// TIA Portal V21 export
FUNCTION "PassiProduzione_010102" : Void   // FC145, LAD
{ S7_Optimized_Access := 'TRUE' }
// stored: SetENOAutomatically false
   VAR_TEMP
      CondizioniPassoEsterne : Bool;
      AbilitazionePasso : Bool;
      AppoggioComando : Int;
      ComandoValvolaB : Int;
      PompaPistoniAbilitata : Bool;
   END_VAR
   VAR CONSTANT
      Positivo : Int := 2;
      Negativo : Int := 3;
      FolleScarico : Int := 4;
      FlipFlop : Int := 5;
      SmettiDiContare : Int := 0;
      ResettaIlConteggio : Int := 1;
      Stop : Int := 6;
   END_VAR
BEGIN

REGION Network 1: Sequenza: Produzione - Passo: Sterilizzazione. Condizioni passo esterne.
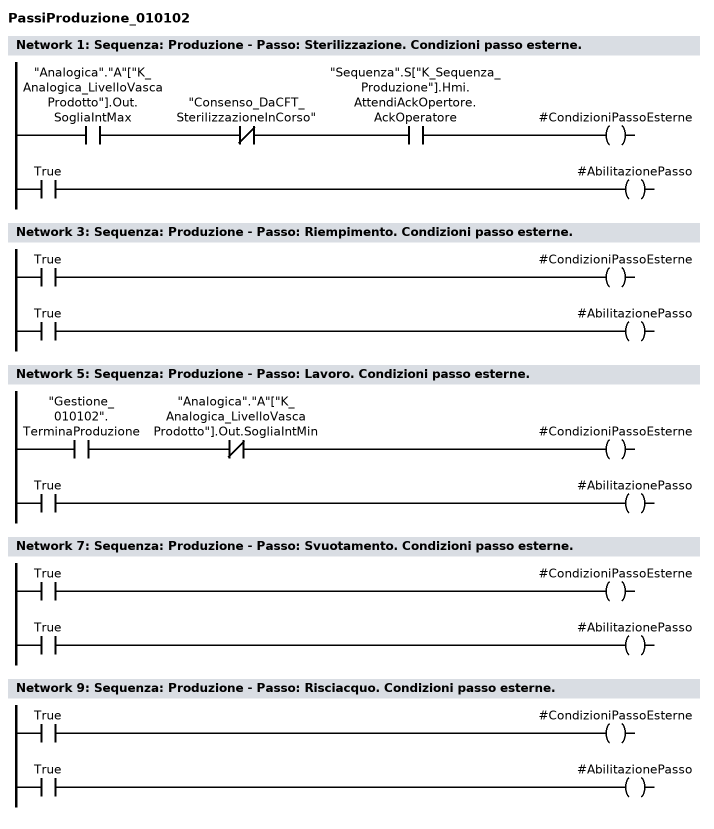
   RUNG wire#powerrail
      Contact( "Analogica"."A"["K_Analogica_LivelloVascaProdotto"].Out.SogliaIntMax )
      I_Contact( "Consenso_DaCFT_SterilizzazioneInCorso" )
      Contact( "Sequenza".S["K_Sequenza_Produzione"].Hmi.AttendiAckOpertore.AckOperatore )
      Coil( #CondizioniPassoEsterne )
   END_RUNG
   RUNG wire#powerrail
      Contact( True )
      Coil( #AbilitazionePasso )
   END_RUNG
   // the same network as SCL:
   #CondizioniPassoEsterne := "Analogica"."A"["K_Analogica_LivelloVascaProdotto"].Out.SogliaIntMax AND NOT "Consenso_DaCFT_SterilizzazioneInCorso" AND "Sequenza".S["K_Sequenza_Produzione"].Hmi.AttendiAckOpertore.AckOperatore;
   #AbilitazionePasso := True;
END_REGION

REGION Network 2 (SCL): Sequenza: Produzione - Passo: Sterilizzazione. Gestione del passo.
   REGION Parametri del passo
       "GestPasso"(K_PassoAttuale := "K_Passo_Sterilizzazione",
                   K_PassoSuccessivo := "K_Passo_Riempimento",
                   AbilitaSaltapasso := True,
                   AbilitaPasso:= #AbilitazionePasso,
                   CondizioniPassoEsterne := #CondizioniPassoEsterne,
                   K_Sequenza := "K_Sequenza_Produzione");
   END_REGION ;
   REGION Comando delle utenze nel passo 
       "GestPasso_CmdValvola"(K_Valvola := "K_Valvola_I",
                              Comando := #Positivo,
                              K_Sequenza := "K_Sequenza_Produzione",
                              K_Passo := "K_Passo_Sterilizzazione",
                              NonAttenderePosizione := False);

       "GestPasso_CmdValvola"(K_Valvola := "K_Valvola_D",
                              Comando := #Positivo,
                              K_Sequenza := "K_Sequenza_Produzione",
                              K_Passo := "K_Passo_Sterilizzazione",
                              NonAttenderePosizione := False);

       "GestPasso_CmdValvola"(K_Valvola := "K_Valvola_D2",
                              Comando := #Positivo,
                              K_Sequenza := "K_Sequenza_Produzione",
                              K_Passo := "K_Passo_Sterilizzazione",
                              NonAttenderePosizione := True);

       "GestPasso_CmdValvola"(K_Valvola := "K_Valvola_B",
                              Comando := #Positivo,
                              K_Sequenza := "K_Sequenza_Produzione",
                              K_Passo := "K_Passo_Sterilizzazione",
                              NonAttenderePosizione := False);

       "GestPasso_CmdValvola"(K_Valvola := "K_Valvola_B1",
                              Comando := "GestPasso_ReplicaComandoValvola"("K_Valvola_B"),
                              K_Sequenza := "K_Sequenza_Produzione",
                              K_Passo := "K_Passo_Sterilizzazione",
                              NonAttenderePosizione := False);

       "GestPasso_CmdValvolaFlipFlop"(K_Valvola := "K_Valvola_L",
                                      NumeroCicli := 1,
                                      TempoPositivo := 1500,
                                      TempoNegativo := 5,
                                      ComandoARiposo := #Negativo,
                                      K_Passo := "K_Passo_Sterilizzazione",
                                      K_Sequenza := "K_Sequenza_Produzione");

       "GestPasso_CmdValvola"(K_Valvola := "K_Valvola_F",
                              Comando := #Positivo,
                              K_Sequenza := "K_Sequenza_Produzione",
                              K_Passo := "K_Passo_Sterilizzazione",
                              NonAttenderePosizione := False);

       "GestPasso_CmdValvola"(K_Valvola := "K_Valvola_CP1",
                              Comando := #Positivo,
                              K_Sequenza := "K_Sequenza_Produzione",
                              K_Passo := "K_Passo_Sterilizzazione",
                              NonAttenderePosizione := False);

       "GestPasso_CmdValvola"(K_Valvola := "K_Valvola_CP2",
                              Comando := #Positivo,
                              K_Sequenza := "K_Sequenza_Produzione",
                              K_Passo := "K_Passo_Sterilizzazione",
                              NonAttenderePosizione := False);

       "GestPasso_AttendiAnalogica"(K_Analogica := "K_Analogica_TemperaturaFineLinea",
                                    KAllAnalog := "KAllAnalog_IntMax",
                                    Comportamento := #ResettaIlConteggio,
                                    K_Sequenza := "K_Sequenza_Produzione",
                                    K_Passo := "K_Passo_Sterilizzazione",
                                    NonAttenderePosizione := False);
       //Motori
       "GestPasso_CmdMotore"(K_Motore := "K_Motore_PompaRicircoloAcquaCalda",
                             Comando := #Positivo,
                             K_Sequenza := "K_Sequenza_Produzione",
                             K_Passo := "K_Passo_Sterilizzazione",
                             NonAttenderePosizione := False);
   END_REGION ;
END_REGION

REGION Network 3: Sequenza: Produzione - Passo: Riempimento. Condizioni passo esterne.
   RUNG wire#powerrail
      Contact( True )
      Coil( #CondizioniPassoEsterne )
   END_RUNG
   RUNG wire#powerrail
      Contact( True )
      Coil( #AbilitazionePasso )
   END_RUNG
   // the same network as SCL:
   #CondizioniPassoEsterne := True;
   #AbilitazionePasso := True;
END_REGION

REGION Network 4 (SCL): Sequenza: Produzione - Passo: Riempimento. Gestione del passo.
   REGION Parametri del passo
       "GestPasso"(K_PassoAttuale := "K_Passo_Riempimento",
                   K_PassoSuccessivo := "K_Passo_Lavoro",
                   AbilitaSaltapasso := True,
                   AbilitaPasso:= #AbilitazionePasso,
                   CondizioniPassoEsterne := #CondizioniPassoEsterne,
                   K_Sequenza := "K_Sequenza_Produzione");
   END_REGION ;
   REGION Comando delle utenze nel passo 

       "GestPasso_CmdValvola"(K_Valvola := "K_Valvola_D",
                              Comando := #Positivo,
                              K_Sequenza := "K_Sequenza_Produzione",
                              K_Passo := "K_Passo_Riempimento",
                              NonAttenderePosizione := False);

       "GestPasso_CmdValvola"(K_Valvola := "K_Valvola_D2",
                              Comando := #Positivo,
                              K_Sequenza := "K_Sequenza_Produzione",
                              K_Passo := "K_Passo_Riempimento",
                              NonAttenderePosizione := False);

       IF "Analogica".A[K_Analogica_TemperaturaUscitaSterilizzatoreProcesso].Out.SogliaIntMin THEN
           #ComandoValvolaB := #Positivo;
       ELSE
           #ComandoValvolaB := #Negativo;
       END_IF;

       "GestPasso_CmdValvola"(K_Valvola := "K_Valvola_R",
                              Comando := #Positivo,
                              K_Sequenza := "K_Sequenza_Produzione",
                              K_Passo := "K_Passo_Riempimento",
                              NonAttenderePosizione := False);

       "GestPasso_CmdValvola"(K_Valvola := "K_Valvola_B",
                              Comando := #ComandoValvolaB,
                              K_Sequenza := "K_Sequenza_Produzione",
                              K_Passo := "K_Passo_Riempimento",
                              NonAttenderePosizione := False);

       "GestPasso_CmdValvola"(K_Valvola := "K_Valvola_B1",
                              Comando := "GestPasso_ReplicaComandoValvola"("K_Valvola_B"),
                              K_Sequenza := "K_Sequenza_Produzione",
                              K_Passo := "K_Passo_Riempimento",
                              NonAttenderePosizione := False);

       "GestPasso_CmdValvola"(K_Valvola := "K_Valvola_CP1",
                              Comando := #Positivo,
                              K_Sequenza := "K_Sequenza_Produzione",
                              K_Passo := "K_Passo_Riempimento",
                              NonAttenderePosizione := False);

       "GestPasso_CmdValvola"(K_Valvola := "K_Valvola_CP2",
                              Comando := #Positivo,
                              K_Sequenza := "K_Sequenza_Produzione",
                              K_Passo := "K_Passo_Riempimento",
                              NonAttenderePosizione := False);

       "GestPasso_AttendiTotalizzatore"(K_Portata := "K_Portata_PortataIngresso",
                                        K_Sequenza := "K_Sequenza_Produzione",
                                        K_Passo := "K_Passo_Riempimento",
                                        NonAttenderePosizione := False,
                                        Preset_Metricubi := "Gestione_010102".MetricubiTubazioneRiempimento);


       //Motori
       "GestPasso_CmdMotore"(K_Motore := "K_Motore_PompaRicircoloAcquaCalda",
                             Comando := #Positivo,
                             K_Sequenza := "K_Sequenza_Produzione",
                             K_Passo := "K_Passo_Riempimento",
                             NonAttenderePosizione := False);

       #PompaPistoniAbilitata := "MacchinaARicetta".M[K_MacchinaARicetta_SterilizzatoreTubo].Lavoro.DatoBool[K_DatoRicettaBool_SterilizzatoreTubo_AbilitazionePompaPistoni];

       IF #PompaPistoniAbilitata THEN
           "GestPasso_CmdMotore"(K_Motore := "K_Motore_PompaPistoni",
                                 Comando := #Positivo,
                                 K_Sequenza := "K_Sequenza_Produzione",
                                 K_Passo := "K_Passo_Riempimento",
                                 NonAttenderePosizione := False);
       END_IF;
       "GestPasso_CmdMotore"(K_Motore := "K_Motore_PompaMono",
                             Comando := #Positivo,
                             K_Sequenza := "K_Sequenza_Produzione",
                             K_Passo := "K_Passo_Riempimento",
                             NonAttenderePosizione := False);
   END_REGION ;
END_REGION

REGION Network 5: Sequenza: Produzione - Passo: Lavoro. Condizioni passo esterne.
   RUNG wire#powerrail
      Contact( "Gestione_010102".TerminaProduzione )
      I_Contact( "Analogica"."A"["K_Analogica_LivelloVascaProdotto"].Out.SogliaIntMin )
      Coil( #CondizioniPassoEsterne )
   END_RUNG
   RUNG wire#powerrail
      Contact( True )
      Coil( #AbilitazionePasso )
   END_RUNG
   // the same network as SCL:
   #CondizioniPassoEsterne := "Gestione_010102".TerminaProduzione AND NOT "Analogica"."A"["K_Analogica_LivelloVascaProdotto"].Out.SogliaIntMin;
   #AbilitazionePasso := True;
END_REGION

REGION Network 6 (SCL): Sequenza: Produzione - Passo: Lavoro. Gestione del passo.
   REGION Parametri del passo
       "GestPasso"(K_PassoAttuale := "K_Passo_Lavoro",
                   K_PassoSuccessivo := "K_Passo_Svuotamento",
                   AbilitaSaltapasso := True,
                   AbilitaPasso:= #AbilitazionePasso,
                   CondizioniPassoEsterne := #CondizioniPassoEsterne,
                   K_Sequenza := "K_Sequenza_Produzione");
   END_REGION ;
   REGION Comando delle utenze nel passo 


       "GestPasso_CmdValvola"(K_Valvola := "K_Valvola_D",
                              Comando := #Positivo,
                              K_Sequenza := "K_Sequenza_Produzione",
                              K_Passo := "K_Passo_Lavoro",
                              NonAttenderePosizione := False);

       "GestPasso_CmdValvola"(K_Valvola := "K_Valvola_D2",
                              Comando := #Positivo,
                              K_Sequenza := "K_Sequenza_Produzione",
                              K_Passo := "K_Passo_Lavoro",
                              NonAttenderePosizione := False);

       IF "Analogica".A[K_Analogica_TemperaturaUscitaSterilizzatoreProcesso].Out.SogliaIntMin THEN

           #ComandoValvolaB := #Positivo;

           "GestPasso_CmdValvola"(K_Valvola := "K_Valvola_X",
                                  Comando := #Positivo,
                                  K_Sequenza := "K_Sequenza_Produzione",
                                  K_Passo := "K_Passo_Lavoro",
                                  NonAttenderePosizione := False);

           "GestPasso_CmdValvola"(K_Valvola := "K_Valvola_D1",
                                  Comando := #Positivo,
                                  K_Sequenza := "K_Sequenza_Produzione",
                                  K_Passo := "K_Passo_Lavoro",
                                  NonAttenderePosizione := False);
       ELSE
           #ComandoValvolaB := #Negativo;
           "GestPasso_CmdValvola"(K_Valvola := "K_Valvola_X2",
                                  Comando := #Positivo,
                                  K_Sequenza := "K_Sequenza_Produzione",
                                  K_Passo := "K_Passo_Lavoro",
                                  NonAttenderePosizione := False);
       END_IF;

       IF NOT "Motore".M[K_Motore_PompaMono].Out.CmdPosMotore THEN
           #ComandoValvolaB := #Negativo;
       END_IF;

       "GestPasso_CmdValvola"(K_Valvola := "K_Valvola_B",
                              Comando := #ComandoValvolaB,
                              K_Sequenza := "K_Sequenza_Produzione",
                              K_Passo := "K_Passo_Lavoro",
                              NonAttenderePosizione := False);

       "GestPasso_CmdValvola"(K_Valvola := "K_Valvola_B1",
                              Comando := "GestPasso_ReplicaComandoValvola"("K_Valvola_B"),
                              K_Sequenza := "K_Sequenza_Produzione",
                              K_Passo := "K_Passo_Lavoro",
                              NonAttenderePosizione := False);

       "GestPasso_CmdValvola"(K_Valvola := "K_Valvola_CP1",
                              Comando := #Positivo,
                              K_Sequenza := "K_Sequenza_Produzione",
                              K_Passo := "K_Passo_Lavoro",
                              NonAttenderePosizione := False);

       "GestPasso_CmdValvola"(K_Valvola := "K_Valvola_CP2",
                              Comando := #Positivo,
                              K_Sequenza := "K_Sequenza_Produzione",
                              K_Passo := "K_Passo_Lavoro",
                              NonAttenderePosizione := False);

       "GestPasso_AttendiTotalizzatore"(K_Portata := "K_Portata_PortataIngresso",
                                        K_Sequenza := "K_Sequenza_Produzione",
                                        K_Passo := "K_Passo_Lavoro",
                                        NonAttenderePosizione := "Gestione_010102".TerminaProduzione,
                                        Preset_Metricubi := "Gestione_010102".MetricubiTubazioneRiempimento);

       //Motori
       IF "Motore".M[K_Motore_PompaMono].Out.CmdPosMotore THEN
           "GestPasso_CmdMotore"(K_Motore := "K_Motore_PompaRicircoloAcquaCalda",
                                 Comando := #Positivo,
                                 K_Sequenza := "K_Sequenza_Produzione",
                                 K_Passo := "K_Passo_Lavoro",
                                 NonAttenderePosizione := False);
       END_IF;
       IF #PompaPistoniAbilitata THEN
           "GestPasso_CmdMotore"(K_Motore := "K_Motore_PompaPistoni",
                                 Comando := #Positivo,
                                 K_Sequenza := "K_Sequenza_Produzione",
                                 K_Passo := "K_Passo_Lavoro",
                                 NonAttenderePosizione := False);
       END_IF;
       "GestPasso_CmdMotore"(K_Motore := "K_Motore_PompaMono",
                             Comando := #Positivo,
                             K_Sequenza := "K_Sequenza_Produzione",
                             K_Passo := "K_Passo_Lavoro",
                             NonAttenderePosizione := False);
   END_REGION ;
END_REGION

REGION Network 7: Sequenza: Produzione - Passo: Svuotamento. Condizioni passo esterne.
   RUNG wire#powerrail
      Contact( True )
      Coil( #CondizioniPassoEsterne )
   END_RUNG
   RUNG wire#powerrail
      Contact( True )
      Coil( #AbilitazionePasso )
   END_RUNG
   // the same network as SCL:
   #CondizioniPassoEsterne := True;
   #AbilitazionePasso := True;
END_REGION

REGION Network 8 (SCL): Sequenza: Produzione - Passo: Svuotamento. Gestione del passo.
   REGION Parametri del passo
       "GestPasso"(K_PassoAttuale := "K_Passo_Svuotamento",
                   K_PassoSuccessivo := "K_Passo_RisciacquoFineSvuotamento",
                   AbilitaSaltapasso := True,
                   AbilitaPasso:= #AbilitazionePasso,
                   CondizioniPassoEsterne := #CondizioniPassoEsterne,
                   K_Sequenza := "K_Sequenza_Produzione");
   END_REGION ;
   REGION Comando delle utenze nel passo 

       "GestPasso_CmdValvola"(K_Valvola := "K_Valvola_D1",
                              Comando := #Positivo,
                              K_Sequenza := "K_Sequenza_Produzione",
                              K_Passo := "K_Passo_Svuotamento",
                              NonAttenderePosizione := False);

       "GestPasso_CmdValvola"(K_Valvola := "K_Valvola_X",
                              Comando := #Positivo,
                              K_Sequenza := "K_Sequenza_Produzione",
                              K_Passo := "K_Passo_Svuotamento",
                              NonAttenderePosizione := False);

       "GestPasso_CmdValvola"(K_Valvola := "K_Valvola_A",
                              Comando := #Positivo,
                              K_Sequenza := "K_Sequenza_Produzione",
                              K_Passo := "K_Passo_Svuotamento",
                              NonAttenderePosizione := "Analogica".A[K_Analogica_LivelloVascaProdotto].Out.SogliaIntMax);

       "GestPasso_CmdValvola"(K_Valvola := "K_Valvola_A1",
                              Comando := #Positivo,
                              K_Sequenza := "K_Sequenza_Produzione",
                              K_Passo := "K_Passo_Svuotamento",
                              NonAttenderePosizione := "Analogica".A[K_Analogica_LivelloVascaProdotto].Out.SogliaIntMax);

       "GestPasso_CmdValvola"(K_Valvola := "K_Valvola_D",
                              Comando := #Positivo,
                              K_Sequenza := "K_Sequenza_Produzione",
                              K_Passo := "K_Passo_Svuotamento",
                              NonAttenderePosizione := False);

       "GestPasso_CmdValvola"(K_Valvola := "K_Valvola_D2",
                              Comando := #Positivo,
                              K_Sequenza := "K_Sequenza_Produzione",
                              K_Passo := "K_Passo_Svuotamento",
                              NonAttenderePosizione := False);



       "GestPasso_CmdValvola"(K_Valvola := "K_Valvola_B",
                              Comando := #Positivo,
                              K_Sequenza := "K_Sequenza_Produzione",
                              K_Passo := "K_Passo_Svuotamento",
                              NonAttenderePosizione := False);

       "GestPasso_CmdValvola"(K_Valvola := "K_Valvola_B1",
                              Comando := "GestPasso_ReplicaComandoValvola"("K_Valvola_B"),
                              K_Sequenza := "K_Sequenza_Produzione",
                              K_Passo := "K_Passo_Svuotamento",
                              NonAttenderePosizione := False);

       "GestPasso_CmdValvola"(K_Valvola := "K_Valvola_CP1",
                              Comando := #Positivo,
                              K_Sequenza := "K_Sequenza_Produzione",
                              K_Passo := "K_Passo_Svuotamento",
                              NonAttenderePosizione := False);

       "GestPasso_CmdValvola"(K_Valvola := "K_Valvola_CP2",
                              Comando := #Positivo,
                              K_Sequenza := "K_Sequenza_Produzione",
                              K_Passo := "K_Passo_Svuotamento",
                              NonAttenderePosizione := False);

       "GestPasso_AttendiTotalizzatore"(K_Portata := "K_Portata_PortataIngresso",
                                        K_Sequenza := "K_Sequenza_Produzione",
                                        K_Passo := "K_Passo_Svuotamento",
                                        NonAttenderePosizione := False,
                                        Preset_Metricubi := "Gestione_010102".MetricubiTubazioneSvuotamento * 2);

       //Motori
       "GestPasso_CmdMotore"(K_Motore := "K_Motore_PompaRicircoloAcquaCalda",
                             Comando := #Positivo,
                             K_Sequenza := "K_Sequenza_Produzione",
                             K_Passo := "K_Passo_Svuotamento",
                             NonAttenderePosizione := False);
       IF #PompaPistoniAbilitata THEN
           "GestPasso_CmdMotore"(K_Motore := "K_Motore_PompaPistoni",
                                 Comando := #Positivo,
                                 K_Sequenza := "K_Sequenza_Produzione",
                                 K_Passo := "K_Passo_Svuotamento",
                                 NonAttenderePosizione := False);
       END_IF;
       "GestPasso_CmdMotore"(K_Motore := "K_Motore_PompaMono",
                             Comando := #Positivo,
                             K_Sequenza := "K_Sequenza_Produzione",
                             K_Passo := "K_Passo_Svuotamento",
                             NonAttenderePosizione := False);
   END_REGION ;
END_REGION

REGION Network 9: Sequenza: Produzione - Passo: Risciacquo. Condizioni passo esterne.
   RUNG wire#powerrail
      Contact( True )
      Coil( #CondizioniPassoEsterne )
   END_RUNG
   RUNG wire#powerrail
      Contact( True )
      Coil( #AbilitazionePasso )
   END_RUNG
   // the same network as SCL:
   #CondizioniPassoEsterne := True;
   #AbilitazionePasso := True;
END_REGION

REGION Network 10 (SCL): Sequenza: Produzione - Passo: Risciacquo. Gestione del passo.
   REGION Parametri del passo
       "GestPasso"(K_PassoAttuale := "K_Passo_RisciacquoFineSvuotamento",
                   K_PassoSuccessivo := 0,
                   AbilitaSaltapasso := True,
                   AbilitaPasso:= #AbilitazionePasso,
                   CondizioniPassoEsterne := #CondizioniPassoEsterne,
                   K_Sequenza := "K_Sequenza_Produzione");
   END_REGION ;
   REGION Comando delle utenze nel passo    

       "GestPasso_CmdValvola"(K_Valvola := "K_Valvola_A",
                              Comando := #Positivo,
                              K_Sequenza := "K_Sequenza_Produzione",
                              K_Passo := "K_Passo_RisciacquoFineSvuotamento",
                              NonAttenderePosizione := "Analogica".A[K_Analogica_LivelloVascaProdotto].Out.SogliaIntMax);

       "GestPasso_CmdValvola"(K_Valvola := "K_Valvola_A1",
                              Comando := #Positivo,
                              K_Sequenza := "K_Sequenza_Produzione",
                              K_Passo := "K_Passo_RisciacquoFineSvuotamento",
                              NonAttenderePosizione := "Analogica".A[K_Analogica_LivelloVascaProdotto].Out.SogliaIntMax);

       "GestPasso_CmdValvola"(K_Valvola := "K_Valvola_B",
                              Comando := #Positivo,
                              K_Sequenza := "K_Sequenza_Produzione",
                              K_Passo := "K_Passo_RisciacquoFineSvuotamento",
                              NonAttenderePosizione := False);

       "GestPasso_CmdValvola"(K_Valvola := "K_Valvola_B1",
                              Comando := "GestPasso_ReplicaComandoValvola"("K_Valvola_B"),
                              K_Sequenza := "K_Sequenza_Produzione",
                              K_Passo := "K_Passo_RisciacquoFineSvuotamento",
                              NonAttenderePosizione := False);

       "GestPasso_CmdValvola"(K_Valvola := "K_Valvola_E",
                              Comando := #Positivo,
                              K_Sequenza := "K_Sequenza_Produzione",
                              K_Passo := "K_Passo_RisciacquoFineSvuotamento",
                              NonAttenderePosizione := False);

       "GestPasso_CmdValvola"(K_Valvola := "K_Valvola_E1",
                              Comando := #Positivo,
                              K_Sequenza := "K_Sequenza_Produzione",
                              K_Passo := "K_Passo_RisciacquoFineSvuotamento",
                              NonAttenderePosizione := False);

       "GestPasso_CmdValvola"(K_Valvola := "K_Valvola_CP1",
                              Comando := #Positivo,
                              K_Sequenza := "K_Sequenza_Produzione",
                              K_Passo := "K_Passo_RisciacquoFineSvuotamento",
                              NonAttenderePosizione := False);

       //Motori
       IF #PompaPistoniAbilitata THEN
           "GestPasso_CmdMotore"(K_Motore := "K_Motore_PompaPistoni",
                                 Comando := #Positivo,
                                 K_Sequenza := "K_Sequenza_Produzione",
                                 K_Passo := "K_Passo_RisciacquoFineSvuotamento",
                                 NonAttenderePosizione := False);
       END_IF;
       "GestPasso_CmdMotore"(K_Motore := "K_Motore_PompaMono",
                             Comando := #Positivo,
                             K_Sequenza := "K_Sequenza_Produzione",
                             K_Passo := "K_Passo_RisciacquoFineSvuotamento",
                             NonAttenderePosizione := False);

       "GestPasso_CmdMotore"(K_Motore := "K_Motore_CentrifugaLavaggio",
                             Comando := #Positivo,
                             K_Sequenza := "K_Sequenza_Produzione",
                             K_Passo := "K_Passo_RisciacquoFineSvuotamento",
                             NonAttenderePosizione := False);

   END_REGION ;
END_REGION
END_FUNCTION
